// TIA Portal V20 export
TYPE "UDT_Service_ParaIndexInfo"
   STRUCT
      ParaIndex : Int;
      ParaType : Int;
   END_STRUCT;
END_TYPE
